{attribute 'qualified_only'}
{attribute 'strict'}
TYPE eGoodUnloadStaState :
( 
	eUnknown,
    eInit,
	eHoming,
	eReady,
	eDwell,
	eProcessing,
	eDepart,
    eError
);
END_TYPE

(* stored: Version 1.1.0.1, ProductVersion 3.1.4020.12
   DUT eGoodUnloadStaState: Id {cfb8c82f-fb4b-48dc-8f5a-02eb8e1c741f} *)
